// TIA Portal V16 export
// export: Created 2022-09-01T14:29:20.3419156Z, ExportSetting WithDefaults, DisplayName Totally Integrated Automation Portal, DisplayVersion V16, DisplayName TIA Portal Version Control Interface, DisplayVersion V16, DisplayName TIA Portal Openness, DisplayVersion V16, DisplayName STEP 7 Professional, DisplayVersion V16, DisplayName STEP 7 Safety, DisplayVersion V16, DisplayName WinCC Advanced, DisplayVersion V16
FUNCTION "Trasfega_Escorridos" : Void   // FC3, LAD
{ S7_Optimized_Access := 'TRUE' }
VERSION : 0.1
// stored: AutoNumber true, IsIECCheckEnabled false, SetENOAutomatically false, UDAEnableTagReadback false
BEGIN

REGION Network 1: Etapa 13 (INÍCIO)
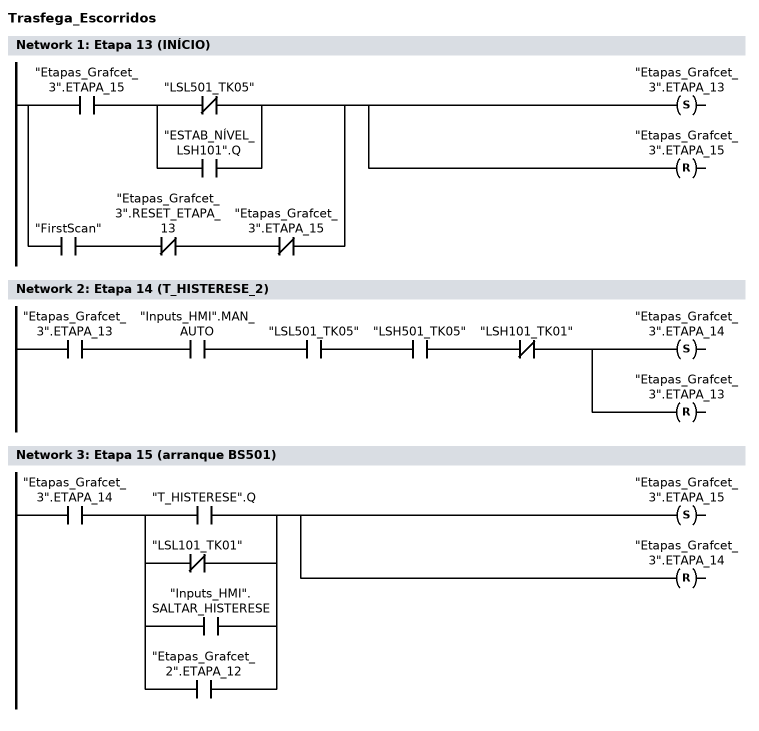
   RUNG wire#powerrail
      Contact( "Etapas_Grafcet_3".ETAPA_15 )
      wire#w1
      I_Contact( "LSL501_TK05" )
      wire#w2
      S_Coil( "Etapas_Grafcet_3".ETAPA_13 )
   END_RUNG
   RUNG wire#w1
      Contact( "ESTAB_NÍVEL_LSH101".Q )
   END_RUNG wire#w2
   RUNG wire#powerrail
      Contact( "FirstScan" )
      I_Contact( "Etapas_Grafcet_3".RESET_ETAPA_13 )
      I_Contact( "Etapas_Grafcet_3".ETAPA_15 )
   END_RUNG wire#w2
   RUNG wire#w2
      R_Coil( "Etapas_Grafcet_3".ETAPA_15 )
   END_RUNG
   // the same network as SCL:
   IF ("Etapas_Grafcet_3".ETAPA_15 AND (NOT "LSL501_TK05" OR "ESTAB_NÍVEL_LSH101".Q)) OR ("FirstScan" AND NOT "Etapas_Grafcet_3".RESET_ETAPA_13 AND NOT "Etapas_Grafcet_3".ETAPA_15) THEN
       "Etapas_Grafcet_3".ETAPA_13 := TRUE;
       "Etapas_Grafcet_3".ETAPA_15 := FALSE;
   END_IF;
END_REGION

REGION Network 2: Etapa 14 (T_HISTERESE_2)
   RUNG wire#powerrail
      Contact( "Etapas_Grafcet_3".ETAPA_13 )
      Contact( "Inputs_HMI".MAN_AUTO )
      Contact( "LSL501_TK05" )
      Contact( "LSH501_TK05" )
      I_Contact( "LSH101_TK01" )
      wire#w1
      S_Coil( "Etapas_Grafcet_3".ETAPA_14 )
   END_RUNG
   RUNG wire#w1
      R_Coil( "Etapas_Grafcet_3".ETAPA_13 )
   END_RUNG
   // the same network as SCL:
   IF "Etapas_Grafcet_3".ETAPA_13 AND "Inputs_HMI".MAN_AUTO AND "LSL501_TK05" AND "LSH501_TK05" AND NOT "LSH101_TK01" THEN
       "Etapas_Grafcet_3".ETAPA_14 := TRUE;
       "Etapas_Grafcet_3".ETAPA_13 := FALSE;
   END_IF;
END_REGION

REGION Network 3: Etapa 15 (arranque BS501)
   RUNG wire#powerrail
      Contact( "Etapas_Grafcet_3".ETAPA_14 )
      wire#w1
      Contact( "T_HISTERESE".Q )
      wire#w2
      S_Coil( "Etapas_Grafcet_3".ETAPA_15 )
   END_RUNG
   RUNG wire#w1
      I_Contact( "LSL101_TK01" )
   END_RUNG wire#w2
   RUNG wire#w1
      Contact( "Inputs_HMI".SALTAR_HISTERESE )
   END_RUNG wire#w2
   RUNG wire#w1
      Contact( "Etapas_Grafcet_2".ETAPA_12 )
   END_RUNG wire#w2
   RUNG wire#w2
      R_Coil( "Etapas_Grafcet_3".ETAPA_14 )
   END_RUNG
   // the same network as SCL:
   IF "Etapas_Grafcet_3".ETAPA_14 AND ("T_HISTERESE".Q OR NOT "LSL101_TK01" OR "Inputs_HMI".SALTAR_HISTERESE OR "Etapas_Grafcet_2".ETAPA_12) THEN
       "Etapas_Grafcet_3".ETAPA_15 := TRUE;
       "Etapas_Grafcet_3".ETAPA_14 := FALSE;
   END_IF;
END_REGION
END_FUNCTION
